(*

short summary
=============
this is the main task of the
candy vending machine application

legal notes
===========
SPDX-FileCopyrightText: © 2024 ekvip automation GmbH <info@ekvip.de>
SPDX-License-Identifier: Apache-2.0
For details check: Apache-2.0_

.. _Apache-2.0: https://www.apache.org/licenses/LICENSE-2.0

*)

PROGRAM MAIN
VAR
	(* to print the log messages with the run method of the logger *)
	loggingProvider :LoggerProvider(0);
	(* behavior for a greedy candy consuming ninja *)
	greedy				:GreedyNinjaCandyBehavior(0);
	(* behavior for a picky candy consuming ninja *)
	picky				:PickyNinjaCandyBehavior(0);
	(* candy preferences of Ajnin *)
	ajninPreferences	:AjninsCandyPreferences();
	(* yeknom as candy consumer *)
	yeknom				:NinjaMonkey(greedy,0);
	(* ajnin as candy consumer *)
	ajnin				:NinjaMonkey(picky, ajninPreferences);
	(* rising edge will feed Ajnin *)
	feedAjnin			:BOOL;
	(* rising edge will feed Yeknom *)
	feedYeknom			:BOOL; 
END_VAR

ajnin.lootCandies(feedAjnin);
yeknom.lootCandies(feedYeknom);
loggingProvider.logger.run();

END_PROGRAM

(* stored: Version 1.1.0.1
   POU MAIN: Id {e86b2847-51a2-4536-ae42-834fd4ee1642}, SpecialFunc None *)
